INTERFACE ITF_MCHMIPrepareScreen_Init EXTENDS ITF_MCHMIPrepareDataForScreen,
	ITF_MCHMIPrepareScreen_00_01_Init, 
	ITF_MCHMIPrepareScreen_00_02_Init,
	ITF_MCHMIPrepareScreen_00_03_Init,
	ITF_MCHMIPrepareScreen_00_04_Init,
	ITF_MCHMIPrepareScreen_00_05_Init,
	ITF_MCHMIPrepareScreen_01_XX_Init,
	ITF_MCHMIPrepareScreen_02_XX_Init,
	ITF_MCHMIPrepareScreen_03_XX_Init,
	ITF_MCHMIPrepareScreen_04_XX_Init,
	ITF_MCHMIPrepareScreen_05_XX_Init,
	ITF_MCHMIPrepareScreen_06_XX_Init,
	ITF_MCHMIPrepareScreen_07_XX_Init,
	ITF_MCHMIPrepareDataForScreenExtension

END_INTERFACE

(* stored: Version 1.1.0.1
   Itf ITF_MCHMIPrepareScreen_Init: Id {0e97142d-a61b-0132-1ba7-e6586d728e01} *)
